// TIA Portal V17 export
// export: Created 2024-09-02T12:50:17.9677419Z, ExportSetting WithDefaults, DisplayName Totally Integrated Automation Portal, DisplayVersion V17, DisplayName TIA Portal Openness, DisplayVersion V17, DisplayName TIA Portal Version Control Interface, DisplayVersion V17, DisplayName STEP 7 Professional, DisplayVersion V17, DisplayName STEP 7 Safety, DisplayVersion V17, DisplayName WinCC Professional, DisplayVersion V17
DATA_BLOCK "AnwDI_CycleTimes_FG02"   // DB1993
{ DB_Accessible_From_OPC_UA := 'FALSE' }
VERSION : 0.1
// stored: AutoNumber false, DBAccessibleFromOPCUA false, InstanceOfName AnwFB_CycleTimes, InstanceOfType FB
"AnwFB_CycleTimes"
   // VAR_INPUT
   //    Start : Bool;
   //    Break : Bool;
   //    Stop : Bool;
   //    Precission : Int;
   // END_VAR
   // VAR_OUTPUT
   //    CycleTimeExceeded : Bool;
   // END_VAR
   // VAR_IN_OUT
   //    CycleTimeIndex : Int;
   //    MainScreenField : DInt;
   //    dataDB : "LTLL_typeData";
   //    configDB : "LTLL_typeConfig";
   // END_VAR
   // VAR
   //    FP : Array[1..16] of Bool;
   //    StartTime : Time;
   //    StartBreakTime : Time;
   //    StopBreakTime : Time;
   //    CurrentBreak : Time;
   //    TotalBreak : Time;
   //    StopTime : Time;
   //    CycleTime : Time;
   //    DIntCycleTime : DWord;
   //    IntCycleTime : Byte;
   //    sPrecission : Int;
   // END_VAR
BEGIN
END_DATA_BLOCK
